PROGRAM Prg_StateMachine
VAR
	Step_0_Init : BOOL;
	Step_1 : BOOL;
	Step_2 : BOOL;
	Step_3: BOOL;
	Step_4 : BOOL;
	
	rTrigA : Tc2_Standard.R_TRIG;
	edgeA : BOOL;
	rTrigB : Tc2_Standard.R_TRIG;
	edgeB : BOOL;
END_VAR

VAR_IN_OUT
	Plant_Ctrl : Udt_PlantControl_Out;
	
	cmSensor2State_sensorA : Udt_CM_Sensor2State;
	cmSensor2State_sensorB : Udt_CM_Sensor2State;
	
	cmActuator3State_ConveyorEntry : Udt_CM_Actuator3State;
	cmActuator3State_ConveyorMain : Udt_CM_Actuator3State;
END_VAR
VAR // added by the converter: edge detectors and wires of the graphical bodies
    _w1, _w2, _w3, _w4 : BOOL;
END_VAR

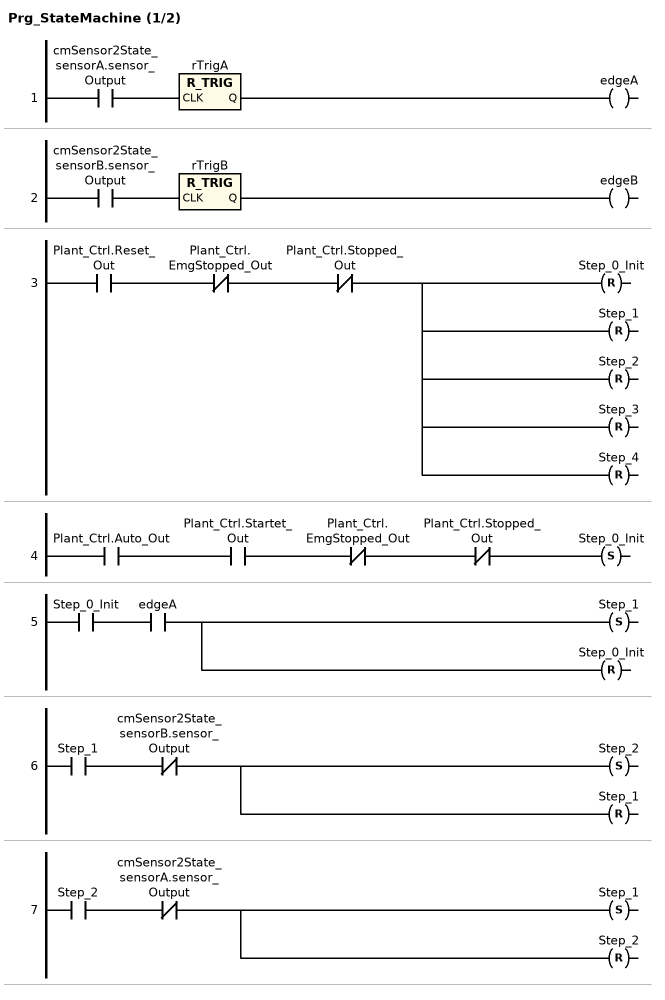
// NETWORK 1
rTrigA(CLK := cmSensor2State_sensorA.sensor_Output); // R_TRIG
edgeA := rTrigA.Q;

// NETWORK 2
rTrigB(CLK := cmSensor2State_sensorB.sensor_Output); // R_TRIG
edgeB := rTrigB.Q;

// NETWORK 3
_w1 := Plant_Ctrl.Reset_Out AND NOT Plant_Ctrl.EmgStopped_Out AND NOT Plant_Ctrl.Stopped_Out;
Step_0_Init R= _w1;
Step_1 R= _w1;
Step_2 R= _w1;
Step_3 R= _w1;
Step_4 R= _w1;

// NETWORK 4
Step_0_Init S= Plant_Ctrl.Auto_Out AND Plant_Ctrl.Startet_Out AND NOT Plant_Ctrl.EmgStopped_Out AND NOT Plant_Ctrl.Stopped_Out;

// NETWORK 5
_w2 := Step_0_Init AND edgeA;
Step_1 S= _w2;
Step_0_Init R= _w2;

// NETWORK 6
_w3 := Step_1 AND NOT cmSensor2State_sensorB.sensor_Output;
Step_2 S= _w3;
Step_1 R= _w3;

// NETWORK 7
_w4 := Step_2 AND NOT cmSensor2State_sensorA.sensor_Output;
Step_1 S= _w4;
Step_2 R= _w4;

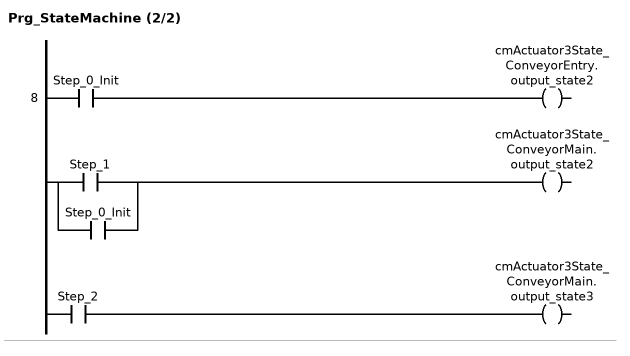
// NETWORK 8
cmActuator3State_ConveyorEntry.output_state2 := Step_0_Init;
cmActuator3State_ConveyorMain.output_state2 := Step_1 OR Step_0_Init;
cmActuator3State_ConveyorMain.output_state3 := Step_2;

END_PROGRAM

(* stored: Version 1.1.0.1, ProductVersion 3.1.4024.13
   POU Prg_StateMachine: Id {a0699d51-4fcb-44af-a102-2c91a55a97d8}, SpecialFunc None *)
